TYPE ST_mcAxisOperationLimits :
STRUCT
	lrSoftMinPosition	:			LREAL;	//Minimum position of travel allowed
	lrSoftMaxPosition	: 			LREAL;	//Maximum position of travel allowed
	lrDefaultAcceleration	:		LREAL;	//Maximum Acceleration allowed
	lrDefaultDeceleration	:		LREAL;	//Minimum deceleration allowed
	lrMaxVelocity		:      		LREAL;  //Maximum Velocity allowed
END_STRUCT
END_TYPE

(* stored: Version 1.1.0.1, ProductVersion 3.1.4024.6
   DUT ST_mcAxisOperationLimits: Id {1279c56f-e78a-46d8-9e11-cc6dfea9d1fa} *)
